TYPE ST_Event :
STRUCT
	eEventType: E_EventType;
END_STRUCT
END_TYPE

(* stored: Version 1.1.0.1, ProductVersion 3.1.4024.16
   DUT ST_Event: Id {976069f4-4b24-40ef-b838-a5d11c09009d} *)
